FUNCTION isLeapYear : BOOL
VAR_INPUT
	Year : DINT;
END_VAR
VAR
END_VAR

isLeapYear := (year mod 4 = 0) and ((year mod 100 <> 0) or (year mod 400 = 0));

END_FUNCTION

(* stored: Version 1.1.0.1, ProductVersion 3.1.4024.12
   POU isLeapYear: Id {5346f763-5f48-48df-8278-4883b2ab8214}, SpecialFunc None *)
